FUNCTION_BLOCK AND_REJECTION (* Composite Function Block Type *)
  (* Standard: 61499-2 *)
  (* Version 0.2, 2003-12-05, JHC, Rockwell Automation, Renamed from NEWCOMPFB. *)
  (* Version 0.1, 2002-01-08, JHC, Rockwell Automation, Added DLY FB as example. *)
  (* Version 0.0, 2000-05-27, JHC, Rockwell Automation *)
  (* Compiler header: package fb.rt.student; *)
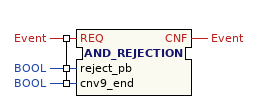
  EVENT_INPUT
    REQ WITH reject_pb, cnv9_end; (* Normal Execution Request *)
  END_EVENT
  EVENT_OUTPUT
    CNF; (* Execution Confirmation *)
  END_EVENT
  VAR_INPUT
    reject_pb : BOOL;
    cnv9_end : BOOL;
  END_VAR
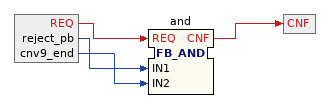
  FBS
    and : FB_AND;
  END_FBS
  EVENT_CONNECTIONS
    REQ TO and.REQ;
    and.CNF TO CNF;
  END_CONNECTIONS
  DATA_CONNECTIONS
    reject_pb TO and.IN1;
    cnv9_end TO and.IN2;
  END_CONNECTIONS
END_FUNCTION_BLOCK
